(* CODESYS project emBRICK_demo_rpi_rs485.project

Project tree, tasks and I/O mapping:
  Device : CODESYS Control for Raspberry Pi MC SL, 3S - Smart Software Solutions GmbH, version 4.0.1.0
    application Application
      libraries: Standard, * (System)
      task MainTask (cyclic, interval t#10ms, priority 1) calls POU
      program POU [ST]
      program POU_ohneMapping [ST]
    CAE_Z_PadBridgeMX : CAE_Z-PatBridgeMX, emBRICK GmbH, order no. VIM0-0204A00, version 1.6
        settings: Communication Type = 2
      CAE_P_2Rel4Di2Ai_01 : CAE_P-2Rel4Di2Ai-01, emBRICK GmbH, order no. VIM0-0150A00, version 1.0
          input  Application.POU.ai_2Rel4Di2Ai[0] :  WORD  // Analog Input 1
          input  Application.POU.ai_2Rel4Di2Ai[1] :  WORD  // Analog Input 2
          input  Application.POU.di_2Rel4Di2Ai[0] : BOOL  // Digital Input.Bit0
          input  Application.POU.di_2Rel4Di2Ai[1] : BOOL  // Digital Input.Bit1
          input  Application.POU.di_2Rel4Di2Ai[2] : BOOL  // Digital Input.Bit2
          input  Application.POU.di_2Rel4Di2Ai[3] : BOOL  // Digital Input.Bit3
          output Application.POU.relais_2Rel4Di2Ai[0] : BOOL  // Relays.Bit0
          output Application.POU.relais_2Rel4Di2Ai[1] : BOOL  // Relays.Bit1
          unmapped channels: Status, Digital Input, Relays
    I²C
    Onewire
    Camera device
      <Empty>
    SoftMotion General Axis Pool
    SPI
    GPIOs_A_B : GPIOs A/B, 3S - Smart Software Solutions GmbH, version 3.5.16.0
        unmapped channels: digital inputs (GPIO0..GPIO31), digital outputs (GPIO0..GPIO31)
  libraries: VisuSymbols, 3.5.10.0 (System)
  text list GlobalTextList
*)

// Device/Application/POU
PROGRAM POU
VAR_INPUT
	// Settings
	callTimeMS : UINT := 10;	// Cycle Time in [ms]	

	// I/Os
	relais_2Rel4Di2Ai : ARRAY[0..1] OF BOOL;
	di_2Rel4Di2Ai : ARRAY[0..3] OF BOOL;
	ai_2Rel4Di2Ai : ARRAY[0..1] OF WORD;
	
	// Helpers
	taskCounter : DWORD := 0;
	oldTaskCounter : DWORD := 0;
END_VAR

taskCounter := taskCounter + 1;
(* - IOs should be updated atleast once every 100ms *)	

// Example Application
	
// Toggle Relais 1 every Second
IF ((taskCounter - oldTaskCounter) * callTimeMS) > 1000 THEN
	IF relais_2Rel4Di2Ai[0] = TRUE THEN
		relais_2Rel4Di2Ai[0] := FALSE;
	ELSE
		relais_2Rel4Di2Ai[0] := TRUE;
	END_IF
	oldTaskCounter := taskCounter;
END_IF

// Switch Relais 2 to Value on Input 1
relais_2Rel4Di2Ai[1] := di_2Rel4Di2Ai[0];

END_PROGRAM

// Device/Application/POU_ohneMapping
PROGRAM POU_ohneMapping
VAR
	// Settings
	callTimeMS : UINT := 10;	// Cycle Time in [ms]
	// Helpers
	taskCounter : DWORD := 0;
	oldTaskCounter : DWORD := 0;
END_VAR

taskCounter := taskCounter + 1;

(* - IOs should be updated once every 100ms *)	

// Example Application
// without Mapping you can Controll your IO's with the variable name and with her Adress
// Relais1 has the Adress %QX0.0
// Relais2 has the Adress %QX0.1
// Toggle Relais 1  every Second
IF ((taskCounter - oldTaskCounter) * callTimeMS) > 1000 THEN
	// Here we take the variable name
	IF Relais1 = TRUE THEN
		// But we can easily work with the adress to
		%QX0.0 := FALSE;
		// Relais1 = TRUE
	ELSE
		Relais1 := TRUE;
	END_IF
	oldTaskCounter := taskCounter;
END_IF

// Switch Relais 2 to Value on Input 1
%QX0.1 := DI1;
//Relais2 := DI1;

END_PROGRAM
